// TIA Portal V20 export
DATA_BLOCK "ModuleService_Setup"   // DB83
TITLE = ServiceControlBlockMediumSetup
{ S7_Optimized_Access := 'TRUE'; DB_Accessible_From_OPC_UA := 'FALSE' }
AUTHOR : Siemens AG
FAMILY : ServiceControl
VERSION : 1.0
// stored: DBAccessibleFromOPCUA false, DBAccessibleFromWebserver false, InstanceOfName UDT_Service_ControlBlockMedium, InstanceOfType UDT
"UDT_Service_ControlBlockMedium"
   // VAR
   //    mode : Int := 2;
   //    stepOrder : "UDT_Service_StepOrderRawDataMedium";
   //    "step" : "UDT_Service_StepRawDataMedium";
   //    procedure : "UDT_Service_ProcedureRawDataMedium";
   //    configurationParameterData : "UDT_Service_ParameterDataMedium";
   //    processValueInData : "UDT_Service_ValueDataMedium";
   //    processValueOutData : "UDT_Service_ValueDataMedium";
   //    reportValueData : "UDT_Service_ValueDataMedium";
   //    serviceInteraction : Array[1..30] of DWord;
   //    plcGuid : String;
   //    serviceGuid : String;
   //    serviceDbNumber : Int;
   // END_VAR
BEGIN
   stepOrder.stepOrder[0..199].stepNumber := -1;
   stepOrder.stepOrder[0..29].stepMonitoringTime := 0;
   stepOrder.stepOrder[0..29].parameter.startIndex := -1;
   stepOrder.stepOrder[0..29].parameter.endIndex := -1;
   stepOrder.parameterIndex[0] := 16#1;
   stepOrder.parameterIndex[1] := 16#0;
   stepOrder.parameterIndex[2] := 16#1;
   "step"."step"[0].command[0] := 16#FFFF_FFFF;
   "step"."step"[1].command[0] := 16#FFFF_FFFF;
   "step"."step"[2].command[0] := 16#FFFF_FFFF;
   "step"."step"[3].command[0] := 16#FFFF_FFFF;
   "step"."step"[4].command[0] := 16#FFFF_FFFF;
   "step"."step"[5].command[0] := 16#FFFF_FFFF;
   "step"."step"[6].command[0] := 16#FFFF_FFFF;
   "step"."step"[7].command[0] := 16#FFFF_FFFF;
   "step"."step"[8].command[0] := 16#FFFF_FFFF;
   "step"."step"[9].command[0] := 16#FFFF_FFFF;
   "step"."step"[10].command[0] := 16#FFFF_FFFF;
   "step"."step"[11].command[0] := 16#FFFF_FFFF;
   "step"."step"[12].command[0] := 16#FFFF_FFFF;
   "step"."step"[13].command[0] := 16#FFFF_FFFF;
   "step"."step"[14].command[0] := 16#FFFF_FFFF;
   "step"."step"[15].command[0] := 16#FFFF_FFFF;
   "step"."step"[16].command[0] := 16#FFFF_FFFF;
   "step"."step"[17].command[0] := 16#FFFF_FFFF;
   "step"."step"[18].command[0] := 16#FFFF_FFFF;
   "step"."step"[19].command[0] := 16#FFFF_FFFF;
   "step"."step"[20].command[0] := 16#FFFF_FFFF;
   "step"."step"[21].command[0] := 16#FFFF_FFFF;
   "step"."step"[22].command[0] := 16#FFFF_FFFF;
   "step"."step"[23].command[0] := 16#FFFF_FFFF;
   "step"."step"[24].command[0] := 16#FFFF_FFFF;
   "step"."step"[25].command[0] := 16#FFFF_FFFF;
   "step"."step"[26].command[0] := 16#FFFF_FFFF;
   "step"."step"[27].command[0] := 16#FFFF_FFFF;
   "step"."step"[28].command[0] := 16#FFFF_FFFF;
   "step"."step"[29].command[0] := 16#FFFF_FFFF;
   "step"."step"[30].command[0] := 16#FFFF_FFFF;
   "step"."step"[31].command[0] := 16#FFFF_FFFF;
   "step"."step"[32].command[0] := 16#FFFF_FFFF;
   "step"."step"[33].command[0] := 16#FFFF_FFFF;
   "step"."step"[34].command[0] := 16#FFFF_FFFF;
   "step"."step"[35].command[0] := 16#FFFF_FFFF;
   "step"."step"[36].command[0] := 16#FFFF_FFFF;
   "step"."step"[37].command[0] := 16#FFFF_FFFF;
   "step"."step"[38].command[0] := 16#FFFF_FFFF;
   "step"."step"[39].command[0] := 16#FFFF_FFFF;
   "step"."step"[40].command[0] := 16#FFFF_FFFF;
   "step"."step"[41].command[0] := 16#FFFF_FFFF;
   "step"."step"[42].command[0] := 16#FFFF_FFFF;
   "step"."step"[43].command[0] := 16#FFFF_FFFF;
   "step"."step"[44].command[0] := 16#FFFF_FFFF;
   "step"."step"[45].command[0] := 16#FFFF_FFFF;
   "step"."step"[46].command[0] := 16#FFFF_FFFF;
   "step"."step"[47].command[0] := 16#FFFF_FFFF;
   "step"."step"[48].command[0] := 16#FFFF_FFFF;
   "step"."step"[49].command[0] := 16#FFFF_FFFF;
   "step"."step"[50].command[0] := 16#FFFF_FFFF;
   "step"."step"[51].command[0] := 16#FFFF_FFFF;
   "step"."step"[52].command[0] := 16#FFFF_FFFF;
   "step"."step"[53].command[0] := 16#FFFF_FFFF;
   "step"."step"[54].command[0] := 16#FFFF_FFFF;
   "step"."step"[55].command[0] := 16#FFFF_FFFF;
   "step"."step"[56].command[0] := 16#FFFF_FFFF;
   "step"."step"[57].command[0] := 16#FFFF_FFFF;
   "step"."step"[58].command[0] := 16#FFFF_FFFF;
   "step"."step"[59].command[0] := 16#FFFF_FFFF;
   "step"."step"[60].command[0] := 16#FFFF_FFFF;
   "step"."step"[61].command[0] := 16#FFFF_FFFF;
   "step"."step"[62].command[0] := 16#FFFF_FFFF;
   "step"."step"[63].command[0] := 16#FFFF_FFFF;
   "step"."step"[64].command[0] := 16#FFFF_FFFF;
   "step"."step"[65].command[0] := 16#FFFF_FFFF;
   "step"."step"[66].command[0] := 16#FFFF_FFFF;
   "step"."step"[67].command[0] := 16#FFFF_FFFF;
   "step"."step"[68].command[0] := 16#FFFF_FFFF;
   "step"."step"[69].command[0] := 16#FFFF_FFFF;
   "step"."step"[70].command[0] := 16#FFFF_FFFF;
   "step"."step"[71].command[0] := 16#FFFF_FFFF;
   "step"."step"[72].command[0] := 16#FFFF_FFFF;
   "step"."step"[73].command[0] := 16#FFFF_FFFF;
   "step"."step"[74].command[0] := 16#FFFF_FFFF;
   "step"."step"[75].command[0] := 16#FFFF_FFFF;
   "step"."step"[76].command[0] := 16#FFFF_FFFF;
   "step"."step"[77].command[0] := 16#FFFF_FFFF;
   "step"."step"[78].command[0] := 16#FFFF_FFFF;
   "step"."step"[79].command[0] := 16#FFFF_FFFF;
   "step"."step"[80].command[0] := 16#FFFF_FFFF;
   "step"."step"[81].command[0] := 16#FFFF_FFFF;
   "step"."step"[82].command[0] := 16#FFFF_FFFF;
   "step"."step"[83].command[0] := 16#FFFF_FFFF;
   "step"."step"[84].command[0] := 16#FFFF_FFFF;
   "step"."step"[85].command[0] := 16#FFFF_FFFF;
   "step"."step"[86].command[0] := 16#FFFF_FFFF;
   "step"."step"[87].command[0] := 16#FFFF_FFFF;
   "step"."step"[88].command[0] := 16#FFFF_FFFF;
   "step"."step"[89].command[0] := 16#FFFF_FFFF;
   "step"."step"[90].command[0] := 16#FFFF_FFFF;
   "step"."step"[91].command[0] := 16#FFFF_FFFF;
   "step"."step"[92].command[0] := 16#FFFF_FFFF;
   "step"."step"[93].command[0] := 16#FFFF_FFFF;
   "step"."step"[94].command[0] := 16#FFFF_FFFF;
   "step"."step"[95].command[0] := 16#FFFF_FFFF;
   "step"."step"[96].command[0] := 16#FFFF_FFFF;
   "step"."step"[97].command[0] := 16#FFFF_FFFF;
   "step"."step"[98].command[0] := 16#FFFF_FFFF;
   "step"."step"[99].command[0] := 16#FFFF_FFFF;
   "step"."step"[0].force[0] := 16#FFFF_FFFF;
   "step"."step"[1].force[0] := 16#FFFF_FFFF;
   "step"."step"[2].force[0] := 16#FFFF_FFFF;
   "step"."step"[3].force[0] := 16#FFFF_FFFF;
   "step"."step"[4].force[0] := 16#FFFF_FFFF;
   "step"."step"[5].force[0] := 16#FFFF_FFFF;
   "step"."step"[6].force[0] := 16#FFFF_FFFF;
   "step"."step"[7].force[0] := 16#FFFF_FFFF;
   "step"."step"[8].force[0] := 16#FFFF_FFFF;
   "step"."step"[9].force[0] := 16#FFFF_FFFF;
   "step"."step"[10].force[0] := 16#FFFF_FFFF;
   "step"."step"[11].force[0] := 16#FFFF_FFFF;
   "step"."step"[12].force[0] := 16#FFFF_FFFF;
   "step"."step"[13].force[0] := 16#FFFF_FFFF;
   "step"."step"[14].force[0] := 16#FFFF_FFFF;
   "step"."step"[15].force[0] := 16#FFFF_FFFF;
   "step"."step"[16].force[0] := 16#FFFF_FFFF;
   "step"."step"[17].force[0] := 16#FFFF_FFFF;
   "step"."step"[18].force[0] := 16#FFFF_FFFF;
   "step"."step"[19].force[0] := 16#FFFF_FFFF;
   "step"."step"[20].force[0] := 16#FFFF_FFFF;
   "step"."step"[21].force[0] := 16#FFFF_FFFF;
   "step"."step"[22].force[0] := 16#FFFF_FFFF;
   "step"."step"[23].force[0] := 16#FFFF_FFFF;
   "step"."step"[24].force[0] := 16#FFFF_FFFF;
   "step"."step"[25].force[0] := 16#FFFF_FFFF;
   "step"."step"[26].force[0] := 16#FFFF_FFFF;
   "step"."step"[27].force[0] := 16#FFFF_FFFF;
   "step"."step"[28].force[0] := 16#FFFF_FFFF;
   "step"."step"[29].force[0] := 16#FFFF_FFFF;
   "step"."step"[30].force[0] := 16#FFFF_FFFF;
   "step"."step"[31].force[0] := 16#FFFF_FFFF;
   "step"."step"[32].force[0] := 16#FFFF_FFFF;
   "step"."step"[33].force[0] := 16#FFFF_FFFF;
   "step"."step"[34].force[0] := 16#FFFF_FFFF;
   "step"."step"[35].force[0] := 16#FFFF_FFFF;
   "step"."step"[36].force[0] := 16#FFFF_FFFF;
   "step"."step"[37].force[0] := 16#FFFF_FFFF;
   "step"."step"[38].force[0] := 16#FFFF_FFFF;
   "step"."step"[39].force[0] := 16#FFFF_FFFF;
   "step"."step"[40].force[0] := 16#FFFF_FFFF;
   "step"."step"[41].force[0] := 16#FFFF_FFFF;
   "step"."step"[42].force[0] := 16#FFFF_FFFF;
   "step"."step"[43].force[0] := 16#FFFF_FFFF;
   "step"."step"[44].force[0] := 16#FFFF_FFFF;
   "step"."step"[45].force[0] := 16#FFFF_FFFF;
   "step"."step"[46].force[0] := 16#FFFF_FFFF;
   "step"."step"[47].force[0] := 16#FFFF_FFFF;
   "step"."step"[48].force[0] := 16#FFFF_FFFF;
   "step"."step"[49].force[0] := 16#FFFF_FFFF;
   "step"."step"[50].force[0] := 16#FFFF_FFFF;
   "step"."step"[51].force[0] := 16#FFFF_FFFF;
   "step"."step"[52].force[0] := 16#FFFF_FFFF;
   "step"."step"[53].force[0] := 16#FFFF_FFFF;
   "step"."step"[54].force[0] := 16#FFFF_FFFF;
   "step"."step"[55].force[0] := 16#FFFF_FFFF;
   "step"."step"[56].force[0] := 16#FFFF_FFFF;
   "step"."step"[57].force[0] := 16#FFFF_FFFF;
   "step"."step"[58].force[0] := 16#FFFF_FFFF;
   "step"."step"[59].force[0] := 16#FFFF_FFFF;
   "step"."step"[60].force[0] := 16#FFFF_FFFF;
   "step"."step"[61].force[0] := 16#FFFF_FFFF;
   "step"."step"[62].force[0] := 16#FFFF_FFFF;
   "step"."step"[63].force[0] := 16#FFFF_FFFF;
   "step"."step"[64].force[0] := 16#FFFF_FFFF;
   "step"."step"[65].force[0] := 16#FFFF_FFFF;
   "step"."step"[66].force[0] := 16#FFFF_FFFF;
   "step"."step"[67].force[0] := 16#FFFF_FFFF;
   "step"."step"[68].force[0] := 16#FFFF_FFFF;
   "step"."step"[69].force[0] := 16#FFFF_FFFF;
   "step"."step"[70].force[0] := 16#FFFF_FFFF;
   "step"."step"[71].force[0] := 16#FFFF_FFFF;
   "step"."step"[72].force[0] := 16#FFFF_FFFF;
   "step"."step"[73].force[0] := 16#FFFF_FFFF;
   "step"."step"[74].force[0] := 16#FFFF_FFFF;
   "step"."step"[75].force[0] := 16#FFFF_FFFF;
   "step"."step"[76].force[0] := 16#FFFF_FFFF;
   "step"."step"[77].force[0] := 16#FFFF_FFFF;
   "step"."step"[78].force[0] := 16#FFFF_FFFF;
   "step"."step"[79].force[0] := 16#FFFF_FFFF;
   "step"."step"[80].force[0] := 16#FFFF_FFFF;
   "step"."step"[81].force[0] := 16#FFFF_FFFF;
   "step"."step"[82].force[0] := 16#FFFF_FFFF;
   "step"."step"[83].force[0] := 16#FFFF_FFFF;
   "step"."step"[84].force[0] := 16#FFFF_FFFF;
   "step"."step"[85].force[0] := 16#FFFF_FFFF;
   "step"."step"[86].force[0] := 16#FFFF_FFFF;
   "step"."step"[87].force[0] := 16#FFFF_FFFF;
   "step"."step"[88].force[0] := 16#FFFF_FFFF;
   "step"."step"[89].force[0] := 16#FFFF_FFFF;
   "step"."step"[90].force[0] := 16#FFFF_FFFF;
   "step"."step"[91].force[0] := 16#FFFF_FFFF;
   "step"."step"[92].force[0] := 16#FFFF_FFFF;
   "step"."step"[93].force[0] := 16#FFFF_FFFF;
   "step"."step"[94].force[0] := 16#FFFF_FFFF;
   "step"."step"[95].force[0] := 16#FFFF_FFFF;
   "step"."step"[96].force[0] := 16#FFFF_FFFF;
   "step"."step"[97].force[0] := 16#FFFF_FFFF;
   "step"."step"[98].force[0] := 16#FFFF_FFFF;
   "step"."step"[99].force[0] := 16#FFFF_FFFF;
   "step"."step"[0].check[0] := 16#FFFF_FFFF;
   "step"."step"[1].check[0] := 16#FFFF_FFFF;
   "step"."step"[2].check[0] := 16#FFFF_FFFF;
   "step"."step"[3].check[0] := 16#FFFF_FFFF;
   "step"."step"[4].check[0] := 16#FFFF_FFFF;
   "step"."step"[5].check[0] := 16#FFFF_FFFF;
   "step"."step"[6].check[0] := 16#FFFF_FFFF;
   "step"."step"[7].check[0] := 16#FFFF_FFFF;
   "step"."step"[8].check[0] := 16#FFFF_FFFF;
   "step"."step"[9].check[0] := 16#FFFF_FFFF;
   "step"."step"[10].check[0] := 16#FFFF_FFFF;
   "step"."step"[11].check[0] := 16#FFFF_FFFF;
   "step"."step"[12].check[0] := 16#FFFF_FFFF;
   "step"."step"[13].check[0] := 16#FFFF_FFFF;
   "step"."step"[14].check[0] := 16#FFFF_FFFF;
   "step"."step"[15].check[0] := 16#FFFF_FFFF;
   "step"."step"[16].check[0] := 16#FFFF_FFFF;
   "step"."step"[17].check[0] := 16#FFFF_FFFF;
   "step"."step"[18].check[0] := 16#FFFF_FFFF;
   "step"."step"[19].check[0] := 16#FFFF_FFFF;
   "step"."step"[20].check[0] := 16#FFFF_FFFF;
   "step"."step"[21].check[0] := 16#FFFF_FFFF;
   "step"."step"[22].check[0] := 16#FFFF_FFFF;
   "step"."step"[23].check[0] := 16#FFFF_FFFF;
   "step"."step"[24].check[0] := 16#FFFF_FFFF;
   "step"."step"[25].check[0] := 16#FFFF_FFFF;
   "step"."step"[26].check[0] := 16#FFFF_FFFF;
   "step"."step"[27].check[0] := 16#FFFF_FFFF;
   "step"."step"[28].check[0] := 16#FFFF_FFFF;
   "step"."step"[29].check[0] := 16#FFFF_FFFF;
   "step"."step"[30].check[0] := 16#FFFF_FFFF;
   "step"."step"[31].check[0] := 16#FFFF_FFFF;
   "step"."step"[32].check[0] := 16#FFFF_FFFF;
   "step"."step"[33].check[0] := 16#FFFF_FFFF;
   "step"."step"[34].check[0] := 16#FFFF_FFFF;
   "step"."step"[35].check[0] := 16#FFFF_FFFF;
   "step"."step"[36].check[0] := 16#FFFF_FFFF;
   "step"."step"[37].check[0] := 16#FFFF_FFFF;
   "step"."step"[38].check[0] := 16#FFFF_FFFF;
   "step"."step"[39].check[0] := 16#FFFF_FFFF;
   "step"."step"[40].check[0] := 16#FFFF_FFFF;
   "step"."step"[41].check[0] := 16#FFFF_FFFF;
   "step"."step"[42].check[0] := 16#FFFF_FFFF;
   "step"."step"[43].check[0] := 16#FFFF_FFFF;
   "step"."step"[44].check[0] := 16#FFFF_FFFF;
   "step"."step"[45].check[0] := 16#FFFF_FFFF;
   "step"."step"[46].check[0] := 16#FFFF_FFFF;
   "step"."step"[47].check[0] := 16#FFFF_FFFF;
   "step"."step"[48].check[0] := 16#FFFF_FFFF;
   "step"."step"[49].check[0] := 16#FFFF_FFFF;
   "step"."step"[50].check[0] := 16#FFFF_FFFF;
   "step"."step"[51].check[0] := 16#FFFF_FFFF;
   "step"."step"[52].check[0] := 16#FFFF_FFFF;
   "step"."step"[53].check[0] := 16#FFFF_FFFF;
   "step"."step"[54].check[0] := 16#FFFF_FFFF;
   "step"."step"[55].check[0] := 16#FFFF_FFFF;
   "step"."step"[56].check[0] := 16#FFFF_FFFF;
   "step"."step"[57].check[0] := 16#FFFF_FFFF;
   "step"."step"[58].check[0] := 16#FFFF_FFFF;
   "step"."step"[59].check[0] := 16#FFFF_FFFF;
   "step"."step"[60].check[0] := 16#FFFF_FFFF;
   "step"."step"[61].check[0] := 16#FFFF_FFFF;
   "step"."step"[62].check[0] := 16#FFFF_FFFF;
   "step"."step"[63].check[0] := 16#FFFF_FFFF;
   "step"."step"[64].check[0] := 16#FFFF_FFFF;
   "step"."step"[65].check[0] := 16#FFFF_FFFF;
   "step"."step"[66].check[0] := 16#FFFF_FFFF;
   "step"."step"[67].check[0] := 16#FFFF_FFFF;
   "step"."step"[68].check[0] := 16#FFFF_FFFF;
   "step"."step"[69].check[0] := 16#FFFF_FFFF;
   "step"."step"[70].check[0] := 16#FFFF_FFFF;
   "step"."step"[71].check[0] := 16#FFFF_FFFF;
   "step"."step"[72].check[0] := 16#FFFF_FFFF;
   "step"."step"[73].check[0] := 16#FFFF_FFFF;
   "step"."step"[74].check[0] := 16#FFFF_FFFF;
   "step"."step"[75].check[0] := 16#FFFF_FFFF;
   "step"."step"[76].check[0] := 16#FFFF_FFFF;
   "step"."step"[77].check[0] := 16#FFFF_FFFF;
   "step"."step"[78].check[0] := 16#FFFF_FFFF;
   "step"."step"[79].check[0] := 16#FFFF_FFFF;
   "step"."step"[80].check[0] := 16#FFFF_FFFF;
   "step"."step"[81].check[0] := 16#FFFF_FFFF;
   "step"."step"[82].check[0] := 16#FFFF_FFFF;
   "step"."step"[83].check[0] := 16#FFFF_FFFF;
   "step"."step"[84].check[0] := 16#FFFF_FFFF;
   "step"."step"[85].check[0] := 16#FFFF_FFFF;
   "step"."step"[86].check[0] := 16#FFFF_FFFF;
   "step"."step"[87].check[0] := 16#FFFF_FFFF;
   "step"."step"[88].check[0] := 16#FFFF_FFFF;
   "step"."step"[89].check[0] := 16#FFFF_FFFF;
   "step"."step"[90].check[0] := 16#FFFF_FFFF;
   "step"."step"[91].check[0] := 16#FFFF_FFFF;
   "step"."step"[92].check[0] := 16#FFFF_FFFF;
   "step"."step"[93].check[0] := 16#FFFF_FFFF;
   "step"."step"[94].check[0] := 16#FFFF_FFFF;
   "step"."step"[95].check[0] := 16#FFFF_FFFF;
   "step"."step"[96].check[0] := 16#FFFF_FFFF;
   "step"."step"[97].check[0] := 16#FFFF_FFFF;
   "step"."step"[98].check[0] := 16#FFFF_FFFF;
   "step"."step"[99].check[0] := 16#FFFF_FFFF;
   "step"."step"[0]."or"[0] := 16#FFFF_FFFF;
   "step"."step"[1]."or"[0] := 16#FFFF_FFFF;
   "step"."step"[2]."or"[0] := 16#FFFF_FFFF;
   "step"."step"[3]."or"[0] := 16#FFFF_FFFF;
   "step"."step"[4]."or"[0] := 16#FFFF_FFFF;
   "step"."step"[5]."or"[0] := 16#FFFF_FFFF;
   "step"."step"[6]."or"[0] := 16#FFFF_FFFF;
   "step"."step"[7]."or"[0] := 16#FFFF_FFFF;
   "step"."step"[8]."or"[0] := 16#FFFF_FFFF;
   "step"."step"[9]."or"[0] := 16#FFFF_FFFF;
   "step"."step"[10]."or"[0] := 16#FFFF_FFFF;
   "step"."step"[11]."or"[0] := 16#FFFF_FFFF;
   "step"."step"[12]."or"[0] := 16#FFFF_FFFF;
   "step"."step"[13]."or"[0] := 16#FFFF_FFFF;
   "step"."step"[14]."or"[0] := 16#FFFF_FFFF;
   "step"."step"[15]."or"[0] := 16#FFFF_FFFF;
   "step"."step"[16]."or"[0] := 16#FFFF_FFFF;
   "step"."step"[17]."or"[0] := 16#FFFF_FFFF;
   "step"."step"[18]."or"[0] := 16#FFFF_FFFF;
   "step"."step"[19]."or"[0] := 16#FFFF_FFFF;
   "step"."step"[20]."or"[0] := 16#FFFF_FFFF;
   "step"."step"[21]."or"[0] := 16#FFFF_FFFF;
   "step"."step"[22]."or"[0] := 16#FFFF_FFFF;
   "step"."step"[23]."or"[0] := 16#FFFF_FFFF;
   "step"."step"[24]."or"[0] := 16#FFFF_FFFF;
   "step"."step"[25]."or"[0] := 16#FFFF_FFFF;
   "step"."step"[26]."or"[0] := 16#FFFF_FFFF;
   "step"."step"[27]."or"[0] := 16#FFFF_FFFF;
   "step"."step"[28]."or"[0] := 16#FFFF_FFFF;
   "step"."step"[29]."or"[0] := 16#FFFF_FFFF;
   "step"."step"[30]."or"[0] := 16#FFFF_FFFF;
   "step"."step"[31]."or"[0] := 16#FFFF_FFFF;
   "step"."step"[32]."or"[0] := 16#FFFF_FFFF;
   "step"."step"[33]."or"[0] := 16#FFFF_FFFF;
   "step"."step"[34]."or"[0] := 16#FFFF_FFFF;
   "step"."step"[35]."or"[0] := 16#FFFF_FFFF;
   "step"."step"[36]."or"[0] := 16#FFFF_FFFF;
   "step"."step"[37]."or"[0] := 16#FFFF_FFFF;
   "step"."step"[38]."or"[0] := 16#FFFF_FFFF;
   "step"."step"[39]."or"[0] := 16#FFFF_FFFF;
   "step"."step"[40]."or"[0] := 16#FFFF_FFFF;
   "step"."step"[41]."or"[0] := 16#FFFF_FFFF;
   "step"."step"[42]."or"[0] := 16#FFFF_FFFF;
   "step"."step"[43]."or"[0] := 16#FFFF_FFFF;
   "step"."step"[44]."or"[0] := 16#FFFF_FFFF;
   "step"."step"[45]."or"[0] := 16#FFFF_FFFF;
   "step"."step"[46]."or"[0] := 16#FFFF_FFFF;
   "step"."step"[47]."or"[0] := 16#FFFF_FFFF;
   "step"."step"[48]."or"[0] := 16#FFFF_FFFF;
   "step"."step"[49]."or"[0] := 16#FFFF_FFFF;
   "step"."step"[50]."or"[0] := 16#FFFF_FFFF;
   "step"."step"[51]."or"[0] := 16#FFFF_FFFF;
   "step"."step"[52]."or"[0] := 16#FFFF_FFFF;
   "step"."step"[53]."or"[0] := 16#FFFF_FFFF;
   "step"."step"[54]."or"[0] := 16#FFFF_FFFF;
   "step"."step"[55]."or"[0] := 16#FFFF_FFFF;
   "step"."step"[56]."or"[0] := 16#FFFF_FFFF;
   "step"."step"[57]."or"[0] := 16#FFFF_FFFF;
   "step"."step"[58]."or"[0] := 16#FFFF_FFFF;
   "step"."step"[59]."or"[0] := 16#FFFF_FFFF;
   "step"."step"[60]."or"[0] := 16#FFFF_FFFF;
   "step"."step"[61]."or"[0] := 16#FFFF_FFFF;
   "step"."step"[62]."or"[0] := 16#FFFF_FFFF;
   "step"."step"[63]."or"[0] := 16#FFFF_FFFF;
   "step"."step"[64]."or"[0] := 16#FFFF_FFFF;
   "step"."step"[65]."or"[0] := 16#FFFF_FFFF;
   "step"."step"[66]."or"[0] := 16#FFFF_FFFF;
   "step"."step"[67]."or"[0] := 16#FFFF_FFFF;
   "step"."step"[68]."or"[0] := 16#FFFF_FFFF;
   "step"."step"[69]."or"[0] := 16#FFFF_FFFF;
   "step"."step"[70]."or"[0] := 16#FFFF_FFFF;
   "step"."step"[71]."or"[0] := 16#FFFF_FFFF;
   "step"."step"[72]."or"[0] := 16#FFFF_FFFF;
   "step"."step"[73]."or"[0] := 16#FFFF_FFFF;
   "step"."step"[74]."or"[0] := 16#FFFF_FFFF;
   "step"."step"[75]."or"[0] := 16#FFFF_FFFF;
   "step"."step"[76]."or"[0] := 16#FFFF_FFFF;
   "step"."step"[77]."or"[0] := 16#FFFF_FFFF;
   "step"."step"[78]."or"[0] := 16#FFFF_FFFF;
   "step"."step"[79]."or"[0] := 16#FFFF_FFFF;
   "step"."step"[80]."or"[0] := 16#FFFF_FFFF;
   "step"."step"[81]."or"[0] := 16#FFFF_FFFF;
   "step"."step"[82]."or"[0] := 16#FFFF_FFFF;
   "step"."step"[83]."or"[0] := 16#FFFF_FFFF;
   "step"."step"[84]."or"[0] := 16#FFFF_FFFF;
   "step"."step"[85]."or"[0] := 16#FFFF_FFFF;
   "step"."step"[86]."or"[0] := 16#FFFF_FFFF;
   "step"."step"[87]."or"[0] := 16#FFFF_FFFF;
   "step"."step"[88]."or"[0] := 16#FFFF_FFFF;
   "step"."step"[89]."or"[0] := 16#FFFF_FFFF;
   "step"."step"[90]."or"[0] := 16#FFFF_FFFF;
   "step"."step"[91]."or"[0] := 16#FFFF_FFFF;
   "step"."step"[92]."or"[0] := 16#FFFF_FFFF;
   "step"."step"[93]."or"[0] := 16#FFFF_FFFF;
   "step"."step"[94]."or"[0] := 16#FFFF_FFFF;
   "step"."step"[95]."or"[0] := 16#FFFF_FFFF;
   "step"."step"[96]."or"[0] := 16#FFFF_FFFF;
   "step"."step"[97]."or"[0] := 16#FFFF_FFFF;
   "step"."step"[98]."or"[0] := 16#FFFF_FFFF;
   "step"."step"[99]."or"[0] := 16#FFFF_FFFF;
   "step".parameterDefinition[0].indexMTP := 0;
   "step".parameterDefinition[1].indexMTP := 1;
   "step".parameterDefinition[0].indexIO := 0;
   "step".parameterDefinition[1].indexIO := 1;
   "step".parameterDefinition[0..1]."type" := 1;
   "step".parameterDefinition[0..31].controlModule := 16#FF;
   procedure.procedure[0..2].Procedure.IsSelfCompleting := True;
   procedure.procedure[3..15].Procedure.IsSelfCompleting := False;
   procedure.procedure[0].Procedure.ProcedureID := 16#1;
   procedure.procedure[1].Procedure.ProcedureID := 16#2;
   procedure.procedure[2].Procedure.ProcedureID := 16#3;
   procedure.procedure[3..15].Procedure.ProcedureID := 16#0;
   procedure.procedure[0..15].Procedure.IsDefault := False;
   procedure.procedure[0..15].StateTransient.starting.startIndex := -1;
   procedure.procedure[0..15].StateTransient.starting.endIndex := -1;
   procedure.procedure[0..15].StateTransient.running.startIndex := -1;
   procedure.procedure[0..15].StateTransient.running.endIndex := -1;
   procedure.procedure[0..15].StateTransient.holding.startIndex := -1;
   procedure.procedure[0..15].StateTransient.holding.endIndex := -1;
   procedure.procedure[0..15].StateTransient.unholding.startIndex := -1;
   procedure.procedure[0..15].StateTransient.unholding.endIndex := -1;
   procedure.procedure[0..15].StateTransient.pausing.startIndex := -1;
   procedure.procedure[0..15].StateTransient.pausing.endIndex := -1;
   procedure.procedure[0..15].StateTransient.resuming.startIndex := -1;
   procedure.procedure[0..15].StateTransient.resuming.endIndex := -1;
   procedure.procedure[0..15].StateTransient.completing.startIndex := -1;
   procedure.procedure[0..15].StateTransient.completing.endIndex := -1;
   procedure.procedure[0..15].StateTransient.stopping.startIndex := -1;
   procedure.procedure[0..15].StateTransient.stopping.endIndex := -1;
   procedure.procedure[0..15].StateTransient.aborting.startIndex := -1;
   procedure.procedure[0..15].StateTransient.aborting.endIndex := -1;
   procedure.procedure[0..15].StateTransient.resetting.startIndex := -1;
   procedure.procedure[0..15].StateTransient.resetting.endIndex := -1;
   procedure.procedure[0].ProcedureReportMap[0] := 16#F;
   procedure.procedure[1].ProcedureReportMap[0] := 16#8;
   procedure.procedure[2].ProcedureReportMap[0] := 16#F;
   procedure.procedure[3].ProcedureReportMap[0] := 16#0;
   procedure.procedure[4].ProcedureReportMap[0] := 16#0;
   procedure.procedure[5].ProcedureReportMap[0] := 16#0;
   procedure.procedure[6].ProcedureReportMap[0] := 16#0;
   procedure.procedure[7].ProcedureReportMap[0] := 16#0;
   procedure.procedure[8].ProcedureReportMap[0] := 16#0;
   procedure.procedure[9].ProcedureReportMap[0] := 16#0;
   procedure.procedure[10].ProcedureReportMap[0] := 16#0;
   procedure.procedure[11].ProcedureReportMap[0] := 16#0;
   procedure.procedure[12].ProcedureReportMap[0] := 16#0;
   procedure.procedure[13].ProcedureReportMap[0] := 16#0;
   procedure.procedure[14].ProcedureReportMap[0] := 16#0;
   procedure.procedure[15].ProcedureReportMap[0] := 16#0;
   procedure.procedure[0].ProcedureProcessInMap[0] := 16#0;
   procedure.procedure[1].ProcedureProcessInMap[0] := 16#0;
   procedure.procedure[2].ProcedureProcessInMap[0] := 16#0;
   procedure.procedure[3].ProcedureProcessInMap[0] := 16#0;
   procedure.procedure[4].ProcedureProcessInMap[0] := 16#0;
   procedure.procedure[5].ProcedureProcessInMap[0] := 16#0;
   procedure.procedure[6].ProcedureProcessInMap[0] := 16#0;
   procedure.procedure[7].ProcedureProcessInMap[0] := 16#0;
   procedure.procedure[8].ProcedureProcessInMap[0] := 16#0;
   procedure.procedure[9].ProcedureProcessInMap[0] := 16#0;
   procedure.procedure[10].ProcedureProcessInMap[0] := 16#0;
   procedure.procedure[11].ProcedureProcessInMap[0] := 16#0;
   procedure.procedure[12].ProcedureProcessInMap[0] := 16#0;
   procedure.procedure[13].ProcedureProcessInMap[0] := 16#0;
   procedure.procedure[14].ProcedureProcessInMap[0] := 16#0;
   procedure.procedure[15].ProcedureProcessInMap[0] := 16#0;
   procedure.procedure[0].ProcedureProcessOutMap[0] := 16#F;
   procedure.procedure[1].ProcedureProcessOutMap[0] := 16#F;
   procedure.procedure[2].ProcedureProcessOutMap[0] := 16#F;
   procedure.procedure[3].ProcedureProcessOutMap[0] := 16#0;
   procedure.procedure[4].ProcedureProcessOutMap[0] := 16#0;
   procedure.procedure[5].ProcedureProcessOutMap[0] := 16#0;
   procedure.procedure[6].ProcedureProcessOutMap[0] := 16#0;
   procedure.procedure[7].ProcedureProcessOutMap[0] := 16#0;
   procedure.procedure[8].ProcedureProcessOutMap[0] := 16#0;
   procedure.procedure[9].ProcedureProcessOutMap[0] := 16#0;
   procedure.procedure[10].ProcedureProcessOutMap[0] := 16#0;
   procedure.procedure[11].ProcedureProcessOutMap[0] := 16#0;
   procedure.procedure[12].ProcedureProcessOutMap[0] := 16#0;
   procedure.procedure[13].ProcedureProcessOutMap[0] := 16#0;
   procedure.procedure[14].ProcedureProcessOutMap[0] := 16#0;
   procedure.procedure[15].ProcedureProcessOutMap[0] := 16#0;
   configurationParameterData.used[0] := 16#0;
   configurationParameterData.definition[0..31].controlModule := 16#FF;
   processValueInData.used[0] := 16#0;
   processValueInData.definition[0..31].controlModule := 16#FF;
   processValueOutData.used[0] := 16#1;
   processValueOutData.definition[0].indexMTP := 8;
   processValueOutData.definition[1].indexMTP := 6;
   processValueOutData.definition[2].indexMTP := 7;
   processValueOutData.definition[3].indexMTP := 9;
   processValueOutData.definition[0].indexIO := 0;
   processValueOutData.definition[1].indexIO := 1;
   processValueOutData.definition[2].indexIO := 2;
   processValueOutData.definition[3].indexIO := 3;
   processValueOutData.definition[0..3]."type" := 1;
   processValueOutData.definition[0..3].controlModule := 16#0;
   processValueOutData.definition[4..31].controlModule := 16#FF;
   reportValueData.used[0] := 16#1;
   reportValueData.definition[0].indexMTP := 1;
   reportValueData.definition[1].indexMTP := 2;
   reportValueData.definition[2].indexMTP := 3;
   reportValueData.definition[3].indexMTP := 8;
   reportValueData.definition[0].indexIO := 0;
   reportValueData.definition[1].indexIO := 1;
   reportValueData.definition[2].indexIO := 2;
   reportValueData.definition[3].indexIO := 3;
   reportValueData.definition[0..3]."type" := 1;
   reportValueData.definition[0..3].controlModule := 16#0;
   reportValueData.definition[4..31].controlModule := 16#FF;
   serviceInteraction[1..30] := 16#0;
END_DATA_BLOCK
